DATA_BLOCK "DB_Robot_Efort"
{ S7_Optimized_Access := 'TRUE' }
VERSION : 0.1
NON_RETAIN
"FB_RobotEfort"

BEGIN

END_DATA_BLOCK

